// TwinCAT 3 PLC project plc
// ProgramVersion: 3.1.4024.0
// libraries:
//   Tc2_Standard, * (Beckhoff Automation GmbH)
//   Tc2_System, * (Beckhoff Automation GmbH)
//   Tc3_Module, * (Beckhoff Automation GmbH)
// project tree:
//   DUTs/ P_Axis_Rx.TcDUT, P_Axis_Tx.TcDUT, T_Axis_Rx.TcDUT, T_Axis_Tx.TcDUT
//   / PlcTask.TcTTO
//   POUs/ MAIN.TcPOU
// real-time tasks:
//   TASK PlcTask: cycle T#2ms, priority 4, ADS port 352
// I/O:
//   DEVICE Device 3 (EtherCAT), AmsNetId 169.254.115.184.4.1
//     Drive 1 (ZeroErr Driver) [ZeroErr Driver]
//     Drive 2 (ZeroErr Driver) [ZeroErr Driver]
//     Drive 3 (ZeroErr Driver) [ZeroErr Driver]
// variable links:
//   plc/plc Instance <-> Device 3 (EtherCAT)/Drive 1 (ZeroErr Driver)
//     PlcTask Inputs/MAIN.P_Axis_1_STATUS/POSITION_VALUE <-> Transmit PDO mapping 0/Position actual value
//     PlcTask Inputs/MAIN.P_Axis_1_STATUS/STATUS_WORD <-> Transmit PDO mapping 0/Status word
//     PlcTask Outputs/MAIN.P_Axis_1_COMMAND/CONTROL_WORD <-> Receive PDO mapping 7/Control word
//     PlcTask Outputs/MAIN.P_Axis_1_COMMAND/MODE_OF_OPERATION <-> Receive PDO mapping 7/Mode of operation
//     PlcTask Outputs/MAIN.P_Axis_1_COMMAND/TARGET_POSIION <-> Receive PDO mapping 7/Target Position
//   plc/plc Instance <-> Device 3 (EtherCAT)/Drive 2 (ZeroErr Driver)
//     PlcTask Inputs/MAIN.P_Axis_2_STATUS/POSITION_VALUE <-> Transmit PDO mapping 0/Position actual value
//     PlcTask Inputs/MAIN.P_Axis_2_STATUS/STATUS_WORD <-> Transmit PDO mapping 0/Status word
//     PlcTask Outputs/MAIN.P_Axis_2_COMMAND/CONTROL_WORD <-> Receive PDO mapping 7/Control word
//     PlcTask Outputs/MAIN.P_Axis_2_COMMAND/MODE_OF_OPERATION <-> Receive PDO mapping 7/Mode of operation
//     PlcTask Outputs/MAIN.P_Axis_2_COMMAND/TARGET_POSIION <-> Receive PDO mapping 7/Target Position
//   plc/plc Instance <-> Device 3 (EtherCAT)/Drive 3 (ZeroErr Driver)
//     PlcTask Inputs/MAIN.T_Axis_1_STATUS/STATUS_WORD <-> Transmit PDO mapping 0/Status word
//     PlcTask Inputs/MAIN.T_Axis_1_STATUS/TORQUE_VALUE <-> Transmit PDO mapping 0/Torque Actual Value
//     PlcTask Outputs/MAIN.T_Axis_1_COMMAND/CONTROL_WORD <-> Receive PDO mapping 8/Controlword
//     PlcTask Outputs/MAIN.T_Axis_1_COMMAND/MAX_MOTOR_SPEED <-> Receive PDO mapping 8/Max motor speed
//     PlcTask Outputs/MAIN.T_Axis_1_COMMAND/MODE_OF_OPERATION <-> Receive PDO mapping 8/Modes of operation
//     PlcTask Outputs/MAIN.T_Axis_1_COMMAND/TARGET_TORQUE <-> Receive PDO mapping 8/Target torque

CONFIGURATION plc
    RESOURCE PLC ON TwinCAT3
        TASK PlcTask(INTERVAL := T#2ms, PRIORITY := 4);
        PROGRAM MAIN WITH PlcTask : MAIN;
    END_RESOURCE
END_CONFIGURATION

// ---- DUTs/P_Axis_Rx.TcDUT
TYPE P_Axis_Rx :
STRUCT
	STATUS_WORD:UINT;
	POSITION_VALUE:DINT;
END_STRUCT
END_TYPE

// ---- DUTs/P_Axis_Tx.TcDUT
TYPE P_Axis_Tx :
STRUCT
	CONTROL_WORD :UINT;
	TARGET_POSIION:DINT;
	MODE_OF_OPERATION:SINT:=1;
END_STRUCT
END_TYPE

// ---- DUTs/T_Axis_Rx.TcDUT
TYPE T_Axis_Rx :
STRUCT
	STATUS_WORD:UINT;
	TORQUE_VALUE:INT;
END_STRUCT
END_TYPE

// ---- DUTs/T_Axis_Tx.TcDUT
TYPE T_Axis_Tx :
STRUCT
	CONTROL_WORD :UINT;
	TARGET_TORQUE:INT;
	MODE_OF_OPERATION:SINT:=4;
	MAX_MOTOR_SPEED : UDINT:=2000000;
END_STRUCT
END_TYPE

// ---- POUs/MAIN.TcPOU
PROGRAM MAIN
VAR
	P_Axis_1_COMMAND AT%QD0:P_Axis_Tx;
	P_Axis_1_STATUS AT%ID0:P_Axis_Rx;
	
	P_Axis_2_COMMAND AT%QD3:P_Axis_Tx;
	P_Axis_2_STATUS AT%ID2:P_Axis_Rx;
	
	T_Axis_1_COMMAND AT%QD100:T_Axis_Tx;
	T_Axis_1_STATUS AT%ID100:T_Axis_Rx;
END_VAR

END_PROGRAM
